INTERFACE I_Error

PROPERTY Error : BOOL
GET
END_GET
END_PROPERTY

PROPERTY ErrorID : UDINT
GET
END_GET
END_PROPERTY

PROPERTY Message : T_MAXSTRING
GET
END_GET
END_PROPERTY

END_INTERFACE

(* stored: Version 1.1.0.1
   Itf I_Error: Id {5274795b-882c-4c0b-bd92-17b71bce3fbe}
   Property Error: Id {cabb6bfb-af24-4545-a54d-84aa04eb4fc9}
   Get Get: Id {68f09782-297f-465a-aa74-00982ac4d2dd}
   Property ErrorID: Id {47a432d2-551b-45b5-a35b-4a8a043fd4f0}
   Get Get: Id {2b14ad2b-77b6-4c09-a5ce-d2ddf23733c7}
   Property Message: Id {c71bd821-916c-460d-a33b-dc974607b25e}
   Get Get: Id {3cb9efde-bc22-4fe8-aa83-67db5ad2a297} *)
